TYPE ST_RuntimeVariableBinding :
STRUCT
	Definition : ST_ConfigVariableInfo;
	NodeHandle : UINT;
END_STRUCT
END_TYPE

(* stored: Version 1.1.0.1, ProductVersion 3.1.4026.18
   DUT ST_RuntimeVariableBinding: Id {174d7b78-0d59-4c4e-a4f7-e18e7eacda5f} *)
